// TIA Portal V18 export
// export: Created 2026-06-08T16:32:20.4539287Z, ExportSetting WithDefaults, DisplayName Totally Integrated Automation Portal, DisplayVersion V18, DisplayName TIA Portal Openness, DisplayVersion V18, DisplayName TIA Portal Version Control Interface, DisplayVersion V18, DisplayName STEP 7 Professional, DisplayVersion V18, DisplayName STEP 7 Safety, DisplayVersion V18, DisplayName WinCC Professional, DisplayVersion V18
FUNCTION_BLOCK "LID PRODUCTION"   // FB2, LAD
VERSION : 0.1
// stored: AutoNumber true, IsIECCheckEnabled false, UDAEnableTagReadback false
BEGIN

REGION Network 1: LID STARTING HANDLE
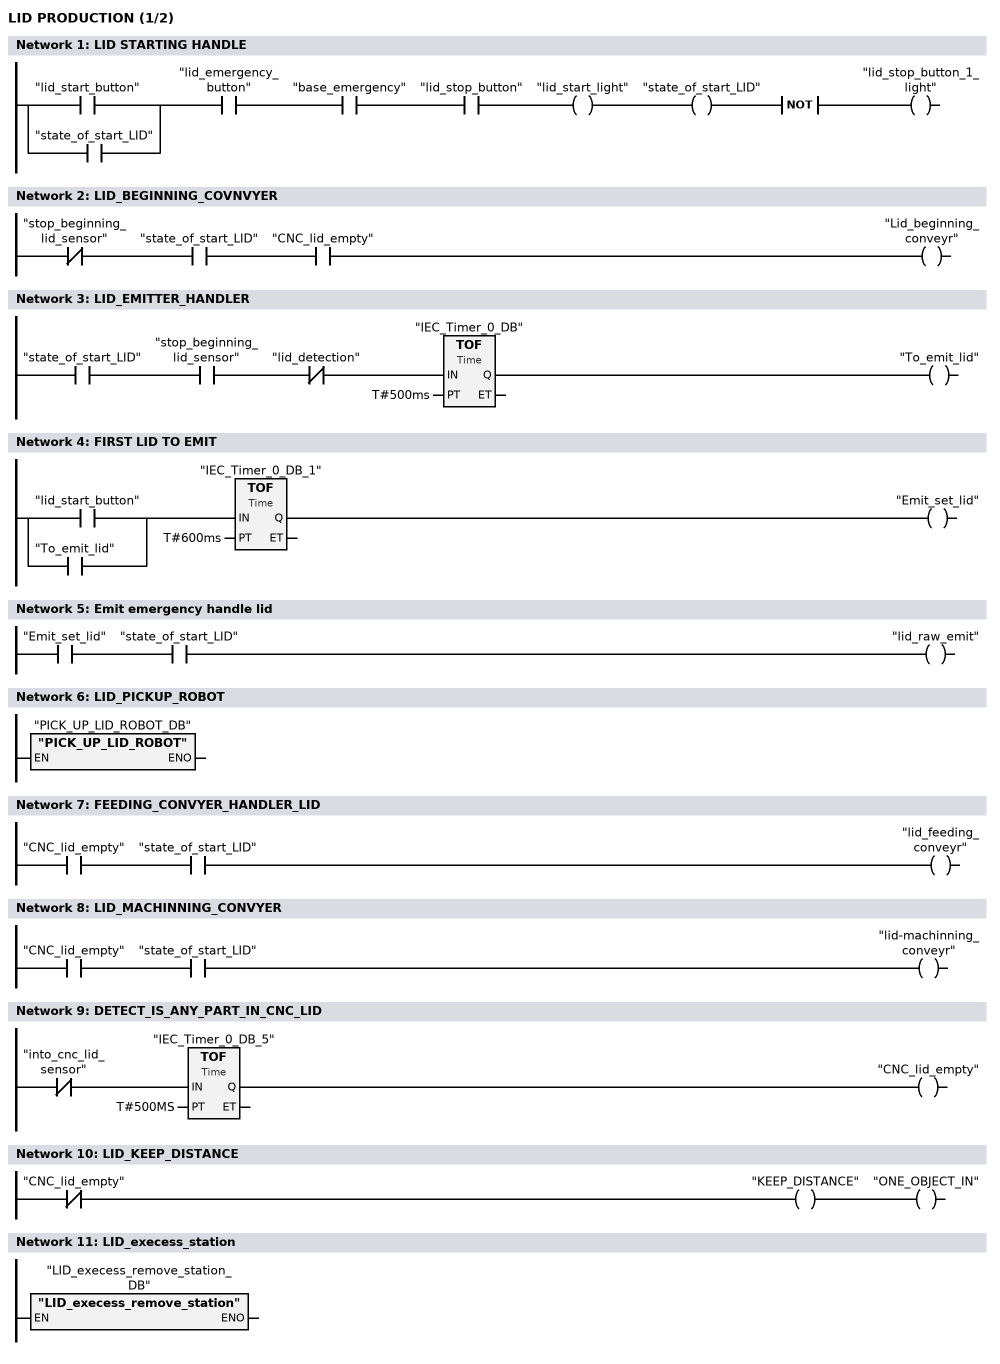
   RUNG wire#powerrail
      Contact( "lid_start_button" )
      wire#w1
      Contact( "lid_emergency_button" )
      Contact( "base_emergency" )
      Contact( "lid_stop_button" )
      Coil( "lid_start_light" )
      Coil( "state_of_start_LID" )
      Not()
      Coil( "lid_stop_button_1_light" )
   END_RUNG
   RUNG wire#powerrail
      Contact( "state_of_start_LID" )
   END_RUNG wire#w1
   // the same network as SCL:
   "lid_start_light" := ("lid_start_button" OR "state_of_start_LID") AND "lid_emergency_button" AND "base_emergency" AND "lid_stop_button";
   "state_of_start_LID" := "lid_start_light";
   "lid_stop_button_1_light" := NOT "lid_start_light";
END_REGION

REGION Network 2: LID_BEGINNING_COVNVYER
   RUNG wire#powerrail
      I_Contact( "stop_beginning_lid_sensor" )
      Contact( "state_of_start_LID" )
      Contact( "CNC_lid_empty" )
      Coil( "Lid_beginning_conveyr" )
   END_RUNG
   // the same network as SCL:
   "Lid_beginning_conveyr" := NOT "stop_beginning_lid_sensor" AND "state_of_start_LID" AND "CNC_lid_empty";
END_REGION

REGION Network 3: LID_EMITTER_HANDLER
   RUNG wire#powerrail
      Contact( "state_of_start_LID" )
      Contact( "stop_beginning_lid_sensor" )
      I_Contact( "lid_detection" )
      { S7_Templates := "time_type := Time" } "IEC_Timer_0_DB".TOF(pt := T#500ms, et =>)
      Coil( "To_emit_lid" )
   END_RUNG
   // the same network as SCL:
   "IEC_Timer_0_DB".TOF(IN := "state_of_start_LID" AND "stop_beginning_lid_sensor" AND NOT "lid_detection",
                        PT := T#500ms);
   "To_emit_lid" := "IEC_Timer_0_DB".Q;
END_REGION

REGION Network 4: FIRST LID TO EMIT
   RUNG wire#powerrail
      Contact( "lid_start_button" )
      wire#w1
      { S7_Templates := "time_type := Time" } "IEC_Timer_0_DB_1".TOF(pt := T#600ms, et =>)
      Coil( "Emit_set_lid" )
   END_RUNG
   RUNG wire#powerrail
      Contact( "To_emit_lid" )
   END_RUNG wire#w1
   // the same network as SCL:
   "IEC_Timer_0_DB_1".TOF(IN := "lid_start_button" OR "To_emit_lid", PT := T#600ms);
   "Emit_set_lid" := "IEC_Timer_0_DB_1".Q;
END_REGION

REGION Network 5: Emit emergency handle lid
   RUNG wire#powerrail
      Contact( "Emit_set_lid" )
      Contact( "state_of_start_LID" )
      Coil( "lid_raw_emit" )
   END_RUNG
   // the same network as SCL:
   "lid_raw_emit" := "Emit_set_lid" AND "state_of_start_LID";
END_REGION

REGION Network 6: LID_PICKUP_ROBOT
   RUNG wire#powerrail
      "PICK_UP_LID_ROBOT_DB"()
   END_RUNG
   // the same network as SCL:
   "PICK_UP_LID_ROBOT_DB"();   // "PICK_UP_LID_ROBOT"
END_REGION

REGION Network 7: FEEDING_CONVYER_HANDLER_LID
   RUNG wire#powerrail
      Contact( "CNC_lid_empty" )
      Contact( "state_of_start_LID" )
      Coil( "lid_feeding_conveyr" )
   END_RUNG
   // the same network as SCL:
   "lid_feeding_conveyr" := "CNC_lid_empty" AND "state_of_start_LID";
END_REGION

REGION Network 8: LID_MACHINNING_CONVYER
   RUNG wire#powerrail
      Contact( "CNC_lid_empty" )
      Contact( "state_of_start_LID" )
      Coil( "lid-machinning_conveyr" )
   END_RUNG
   // the same network as SCL:
   "lid-machinning_conveyr" := "CNC_lid_empty" AND "state_of_start_LID";
END_REGION

REGION Network 9: DETECT_IS_ANY_PART_IN_CNC_LID
   RUNG wire#powerrail
      I_Contact( "into_cnc_lid_sensor" )
      { S7_Templates := "time_type := Time" } "IEC_Timer_0_DB_5".TOF(pt := T#500MS, et =>)
      Coil( "CNC_lid_empty" )
   END_RUNG
   // the same network as SCL:
   "IEC_Timer_0_DB_5".TOF(IN := NOT "into_cnc_lid_sensor", PT := T#500MS);
   "CNC_lid_empty" := "IEC_Timer_0_DB_5".Q;
END_REGION

REGION Network 10: LID_KEEP_DISTANCE
   RUNG wire#powerrail
      I_Contact( "CNC_lid_empty" )
      Coil( "KEEP_DISTANCE" )
      Coil( "ONE_OBJECT_IN" )
   END_RUNG
   // the same network as SCL:
   "KEEP_DISTANCE" := NOT "CNC_lid_empty";
   "ONE_OBJECT_IN" := NOT "CNC_lid_empty";
END_REGION

REGION Network 11: LID_execess_station
   RUNG wire#powerrail
      "LID_execess_remove_station_DB"()
   END_RUNG
   // the same network as SCL:
   "LID_execess_remove_station_DB"();   // "LID_execess_remove_station"
END_REGION

REGION Network 12: CNC
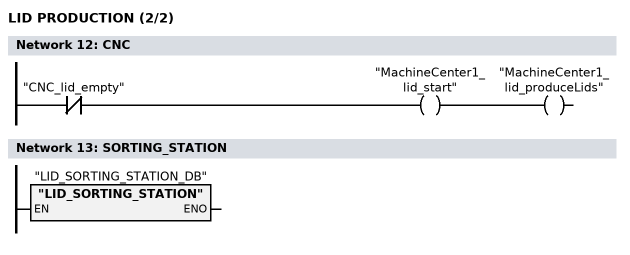
   RUNG wire#powerrail
      I_Contact( "CNC_lid_empty" )
      Coil( "MachineCenter1_lid_start" )
      Coil( "MachineCenter1_lid_produceLids" )
   END_RUNG
   // the same network as SCL:
   "MachineCenter1_lid_start" := NOT "CNC_lid_empty";
   "MachineCenter1_lid_produceLids" := NOT "CNC_lid_empty";
END_REGION

REGION Network 13: SORTING_STATION
   RUNG wire#powerrail
      "LID_SORTING_STATION_DB"()
   END_RUNG
   // the same network as SCL:
   "LID_SORTING_STATION_DB"();   // "LID_SORTING_STATION"
END_REGION
END_FUNCTION_BLOCK
